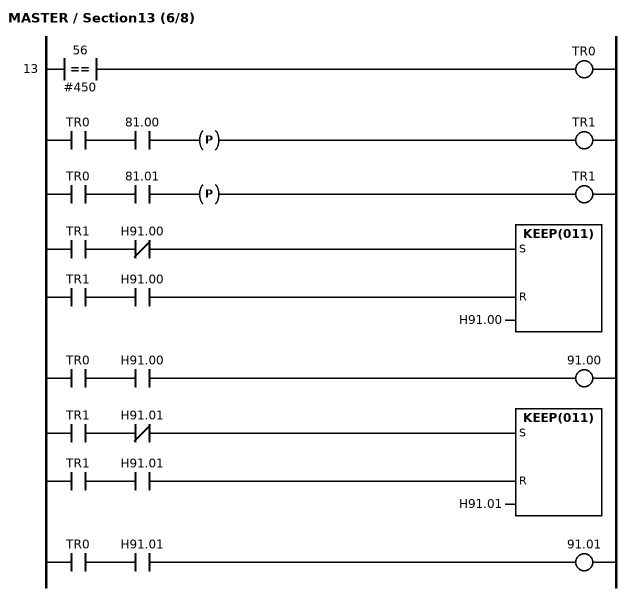
; [picture p48: MASTER / Section13, rungs 13-13]
; rung 13
LD=(300) 56 #450
OUT TR0
AND 81.00
UP(521)
OUT TR1
ANDNOT H91.00
LD TR1
AND H91.00
KEEP(011) H91.00
LD TR0
AND H91.00
OUT 91.00
LD TR0
AND 81.01
UP(521)
OUT TR1
ANDNOT H91.01
LD TR1
AND H91.01
KEEP(011) H91.01
LD TR0
AND H91.01
OUT 91.01

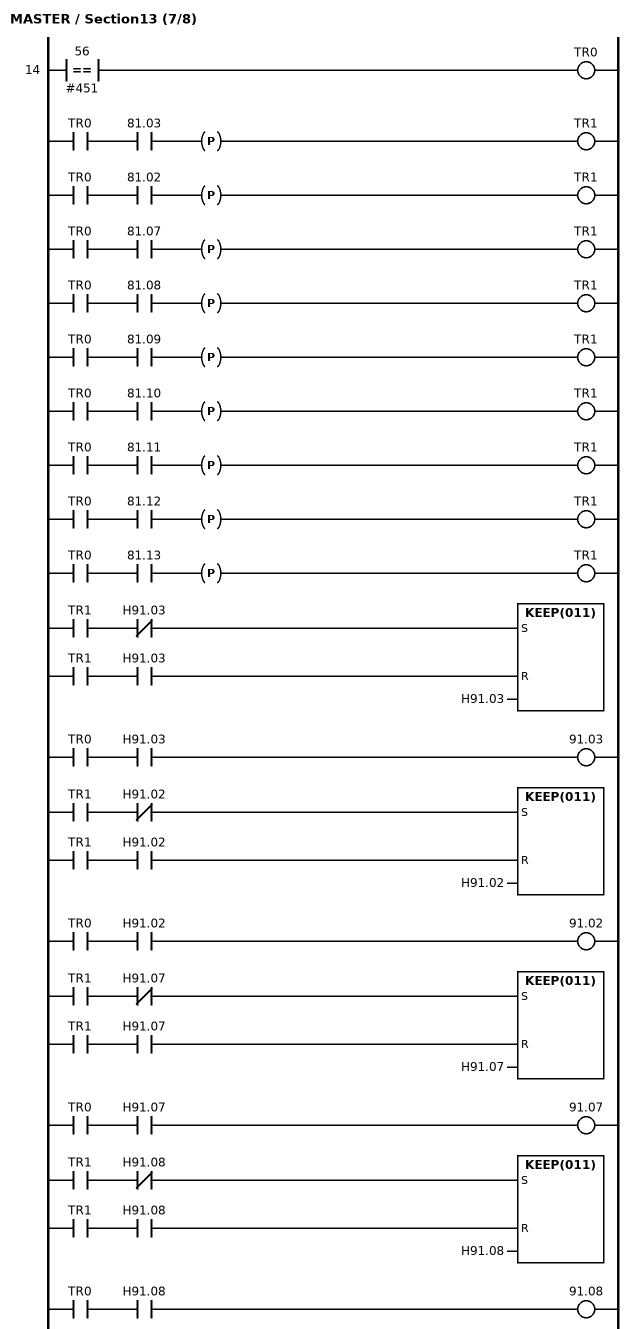

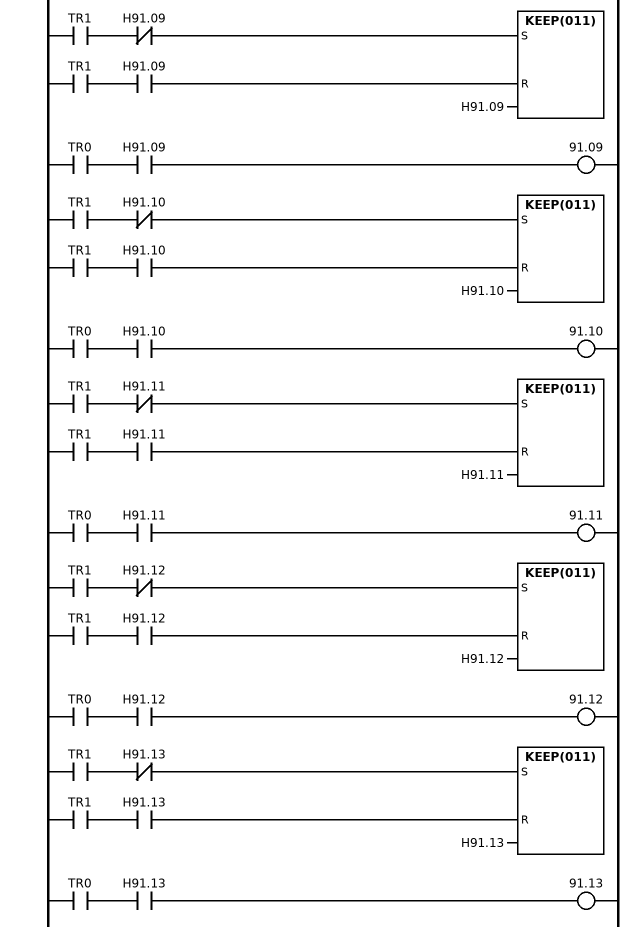
; rung 14
LD=(300) 56 #451
OUT TR0
AND 81.03
UP(521)
OUT TR1
ANDNOT H91.03
LD TR1
AND H91.03
KEEP(011) H91.03
LD TR0
AND H91.03
OUT 91.03
LD TR0
AND 81.02
UP(521)
OUT TR1
ANDNOT H91.02
LD TR1
AND H91.02
KEEP(011) H91.02
LD TR0
AND H91.02
OUT 91.02
LD TR0
AND 81.07
UP(521)
OUT TR1
ANDNOT H91.07
LD TR1
AND H91.07
KEEP(011) H91.07
LD TR0
AND H91.07
OUT 91.07
LD TR0
AND 81.08
UP(521)
OUT TR1
ANDNOT H91.08
LD TR1
AND H91.08
KEEP(011) H91.08
LD TR0
AND H91.08
OUT 91.08
LD TR0
AND 81.09
UP(521)
OUT TR1
ANDNOT H91.09
LD TR1
AND H91.09
KEEP(011) H91.09
LD TR0
AND H91.09
OUT 91.09
LD TR0
AND 81.10
UP(521)
OUT TR1
ANDNOT H91.10
LD TR1
AND H91.10
KEEP(011) H91.10
LD TR0
AND H91.10
OUT 91.10
LD TR0
AND 81.11
UP(521)
OUT TR1
ANDNOT H91.11
LD TR1
AND H91.11
KEEP(011) H91.11
LD TR0
AND H91.11
OUT 91.11
LD TR0
AND 81.12
UP(521)
OUT TR1
ANDNOT H91.12
LD TR1
AND H91.12
KEEP(011) H91.12
LD TR0
AND H91.12
OUT 91.12
LD TR0
AND 81.13
UP(521)
OUT TR1
ANDNOT H91.13
LD TR1
AND H91.13
KEEP(011) H91.13
LD TR0
AND H91.13
OUT 91.13

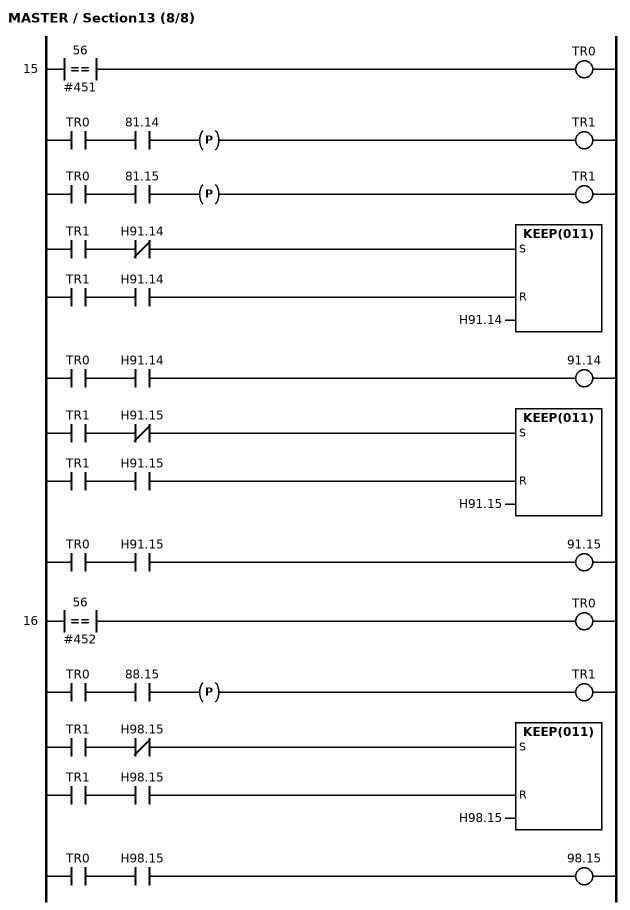
; rung 15
LD=(300) 56 #451
OUT TR0
AND 81.14
UP(521)
OUT TR1
ANDNOT H91.14
LD TR1
AND H91.14
KEEP(011) H91.14
LD TR0
AND H91.14
OUT 91.14
LD TR0
AND 81.15
UP(521)
OUT TR1
ANDNOT H91.15
LD TR1
AND H91.15
KEEP(011) H91.15
LD TR0
AND H91.15
OUT 91.15
; rung 16
LD=(300) 56 #452
OUT TR0
AND 88.15
UP(521)
OUT TR1
ANDNOT H98.15
LD TR1
AND H98.15
KEEP(011) H98.15
LD TR0
AND H98.15
OUT 98.15

### Section Section14

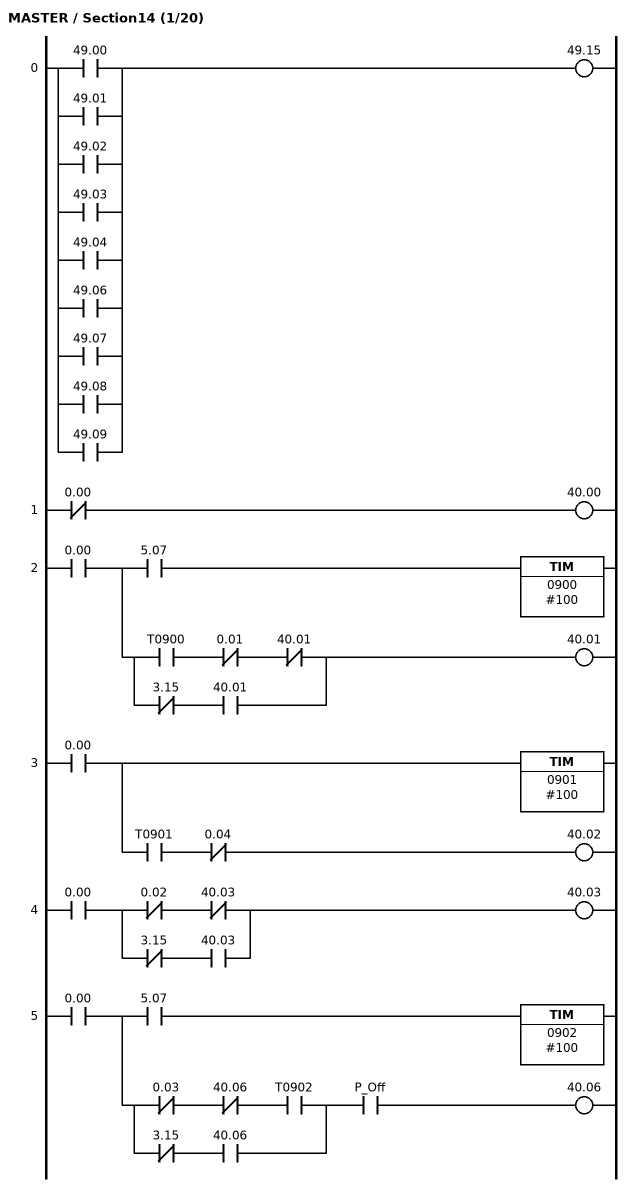
; rung 0
// R
LD 49.00
OR 49.01
OR 49.02
OR 49.03
OR 49.04
OR 49.06
OR 49.07
OR 49.08
OR 49.09
OUT 49.15
; rung 1
// R
LDNOT 0.00
OUT 40.00
; rung 2
// R
LD 0.00
OUT TR0
AND 5.07
TIM 0900 #100
LD TR0
LD T0900
ANDNOT 0.01
ANDNOT 40.01
LDNOT 3.15
AND 40.01
ORLD
ANDLD
OUT 40.01
; rung 3
// R
LD 0.00
TIM 0901 #100
AND T0901
ANDNOT 0.04
OUT 40.02
; rung 4
// R
LD 0.00
LDNOT 0.02
ANDNOT 40.03
LDNOT 3.15
AND 40.03
ORLD
ANDLD
OUT 40.03
; rung 5
// R
LD 0.00
OUT TR0
AND 5.07
TIM 0902 #100
LD TR0
LDNOT 0.03
ANDNOT 40.06
AND T0902
LDNOT 3.15
AND 40.06
ORLD
AND P_Off
ANDLD
OUT 40.06

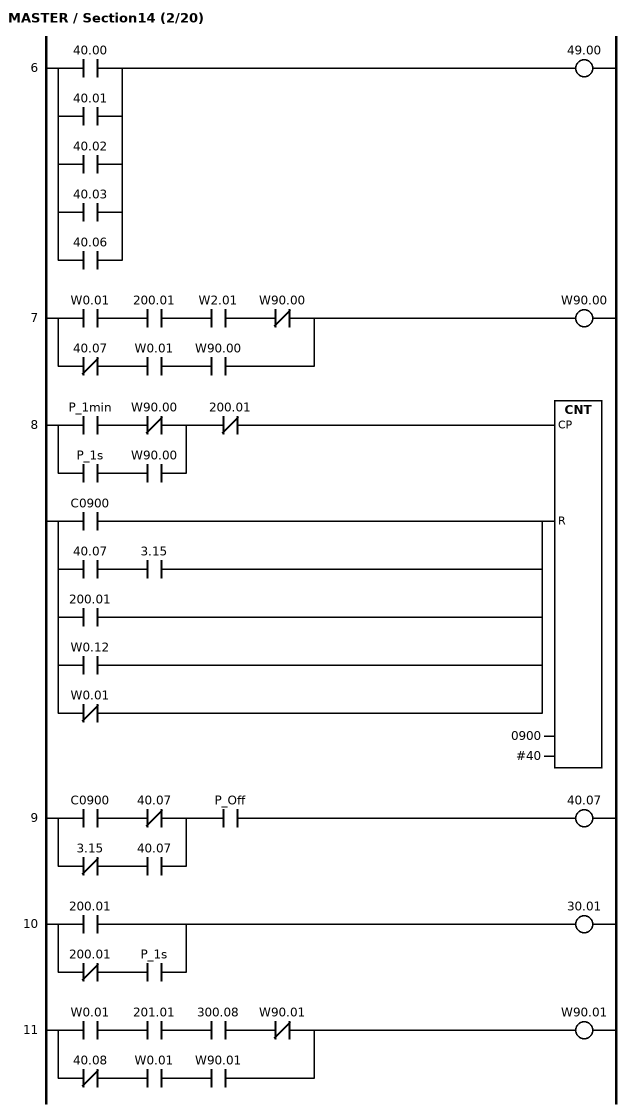
; rung 6
// R
LD 40.00
OR 40.01
OR 40.02
OR 40.03
OR 40.06
OUT 49.00
; rung 7
// R
LD W0.01
AND 200.01
AND W2.01
ANDNOT W90.00
LDNOT 40.07
AND W0.01
AND W90.00
ORLD
OUT W90.00
; rung 8
LD P_1min
ANDNOT W90.00
LD P_1s
AND W90.00
ORLD
ANDNOT 200.01
LD C0900
LD 40.07
AND 3.15
ORLD
OR 200.01
OR W0.12
ORNOT W0.01
CNT 0900 #40
; rung 9
LD C0900
ANDNOT 40.07
LDNOT 3.15
AND 40.07
ORLD
AND P_Off
OUT 40.07
; rung 10
LD 200.01
LDNOT 200.01
AND P_1s
ORLD
OUT 30.01
; rung 11
// R
LD W0.01
AND 201.01
AND 300.08
ANDNOT W90.01
LDNOT 40.08
AND W0.01
AND W90.01
ORLD
OUT W90.01

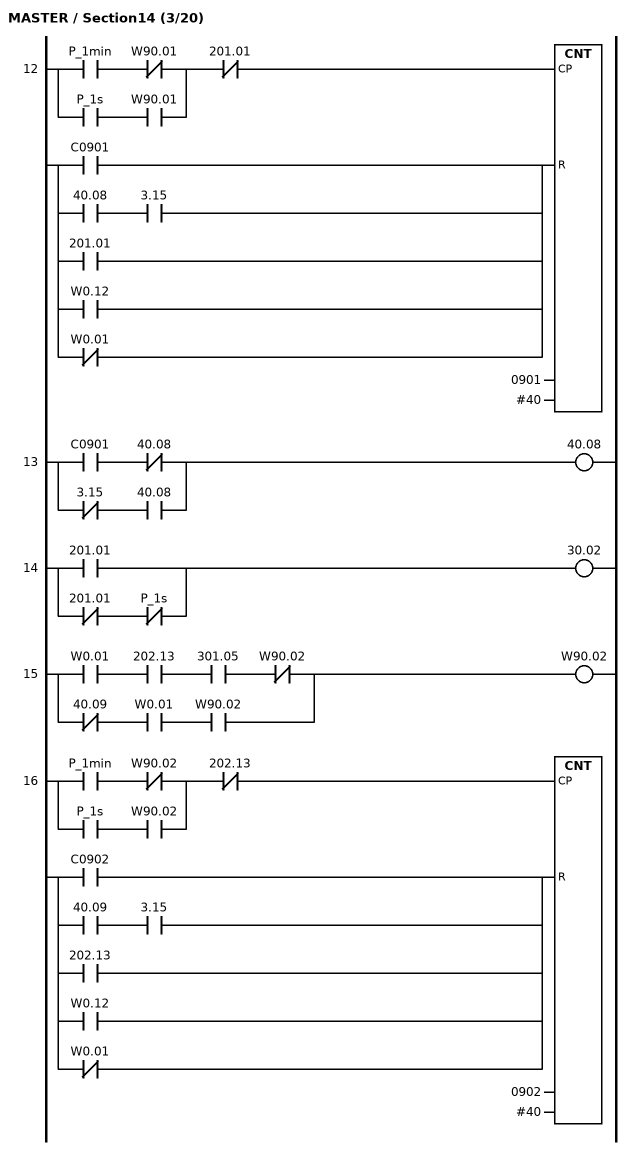
; rung 12
LD P_1min
ANDNOT W90.01
LD P_1s
AND W90.01
ORLD
ANDNOT 201.01
LD C0901
LD 40.08
AND 3.15
ORLD
OR 201.01
OR W0.12
ORNOT W0.01
CNT 0901 #40
; rung 13
LD C0901
ANDNOT 40.08
LDNOT 3.15
AND 40.08
ORLD
OUT 40.08
; rung 14
LD 201.01
LDNOT 201.01
ANDNOT P_1s
ORLD
OUT 30.02
; rung 15
// R
LD W0.01
AND 202.13
AND 301.05
ANDNOT W90.02
LDNOT 40.09
AND W0.01
AND W90.02
ORLD
OUT W90.02
; rung 16
LD P_1min
ANDNOT W90.02
LD P_1s
AND W90.02
ORLD
ANDNOT 202.13
LD C0902
LD 40.09
AND 3.15
ORLD
OR 202.13
OR W0.12
ORNOT W0.01
CNT 0902 #40

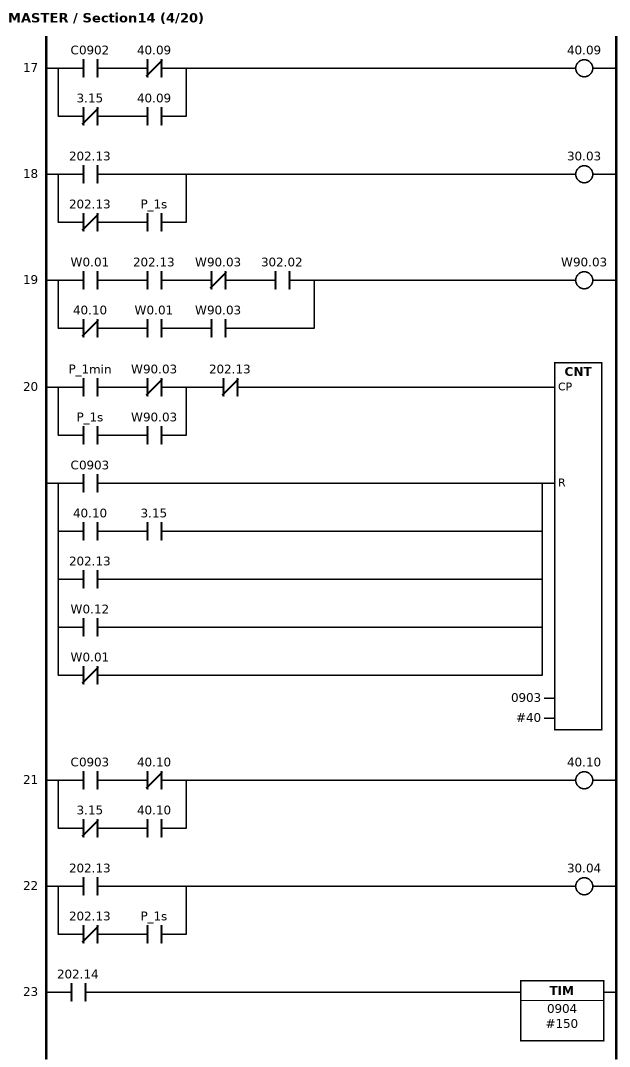
; rung 17
LD C0902
ANDNOT 40.09
LDNOT 3.15
AND 40.09
ORLD
OUT 40.09
; rung 18
LD 202.13
LDNOT 202.13
AND P_1s
ORLD
OUT 30.03
; rung 19
// R
LD W0.01
AND 202.13
ANDNOT W90.03
AND 302.02
LDNOT 40.10
AND W0.01
AND W90.03
ORLD
OUT W90.03
; rung 20
LD P_1min
ANDNOT W90.03
LD P_1s
AND W90.03
ORLD
ANDNOT 202.13
LD C0903
LD 40.10
AND 3.15
ORLD
OR 202.13
OR W0.12
ORNOT W0.01
CNT 0903 #40
; rung 21
LD C0903
ANDNOT 40.10
LDNOT 3.15
AND 40.10
ORLD
OUT 40.10
; rung 22
LD 202.13
LDNOT 202.13
AND P_1s
ORLD
OUT 30.04
; rung 23
LD 202.14
TIM 0904 #150

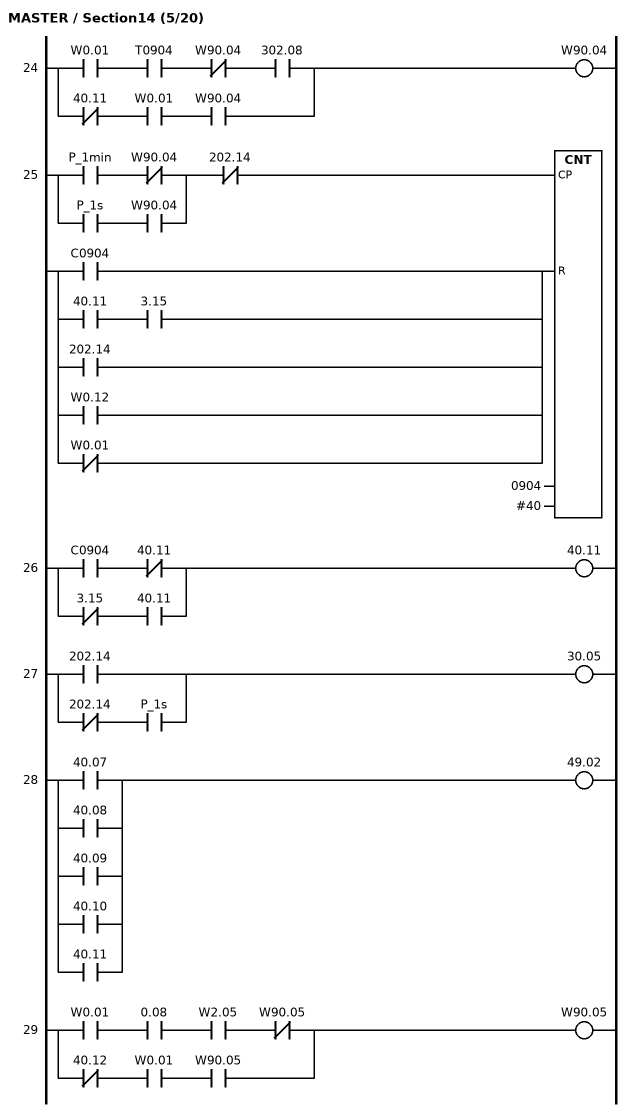
; rung 24
// R
LD W0.01
AND T0904
ANDNOT W90.04
AND 302.08
LDNOT 40.11
AND W0.01
AND W90.04
ORLD
OUT W90.04
; rung 25
LD P_1min
ANDNOT W90.04
LD P_1s
AND W90.04
ORLD
ANDNOT 202.14
LD C0904
LD 40.11
AND 3.15
ORLD
OR 202.14
OR W0.12
ORNOT W0.01
CNT 0904 #40
; rung 26
LD C0904
ANDNOT 40.11
LDNOT 3.15
AND 40.11
ORLD
OUT 40.11
; rung 27
LD 202.14
LDNOT 202.14
AND P_1s
ORLD
OUT 30.05
; rung 28
LD 40.07
OR 40.08
OR 40.09
OR 40.10
OR 40.11
OUT 49.02
; rung 29
// R
LD W0.01
AND 0.08
AND W2.05
ANDNOT W90.05
LDNOT 40.12
AND W0.01
AND W90.05
ORLD
OUT W90.05

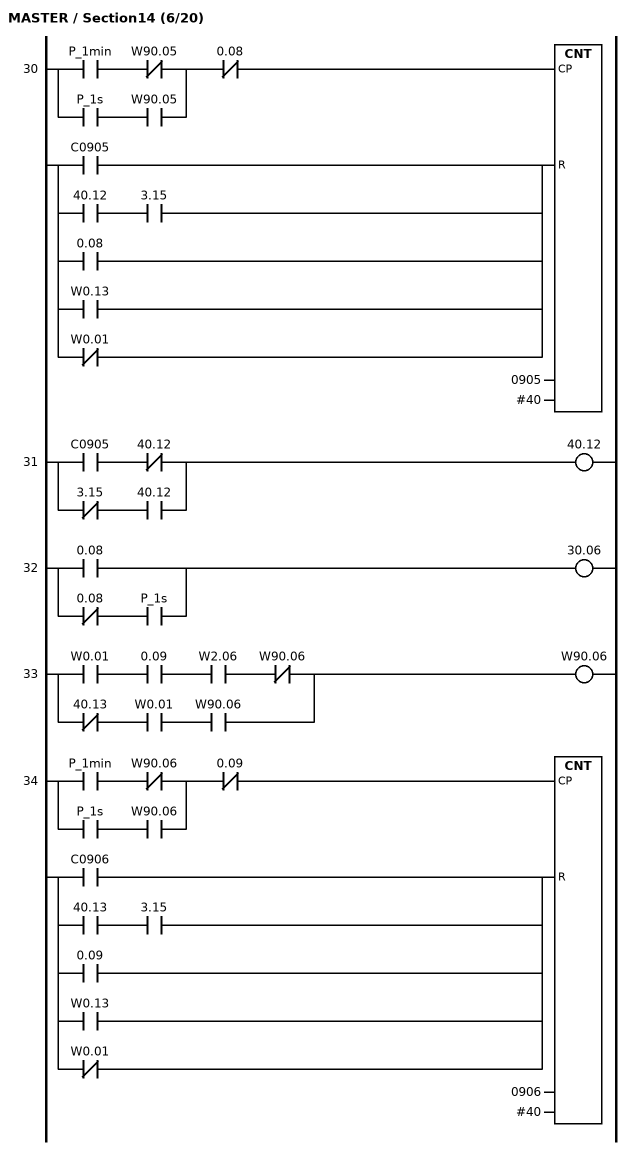
; rung 30
LD P_1min
ANDNOT W90.05
LD P_1s
AND W90.05
ORLD
ANDNOT 0.08
LD C0905
LD 40.12
AND 3.15
ORLD
OR 0.08
OR W0.13
ORNOT W0.01
CNT 0905 #40
; rung 31
LD C0905
ANDNOT 40.12
LDNOT 3.15
AND 40.12
ORLD
OUT 40.12
; rung 32
LD 0.08
LDNOT 0.08
AND P_1s
ORLD
OUT 30.06
; rung 33
// R
LD W0.01
AND 0.09
AND W2.06
ANDNOT W90.06
LDNOT 40.13
AND W0.01
AND W90.06
ORLD
OUT W90.06
; rung 34
LD P_1min
ANDNOT W90.06
LD P_1s
AND W90.06
ORLD
ANDNOT 0.09
LD C0906
LD 40.13
AND 3.15
ORLD
OR 0.09
OR W0.13
ORNOT W0.01
CNT 0906 #40

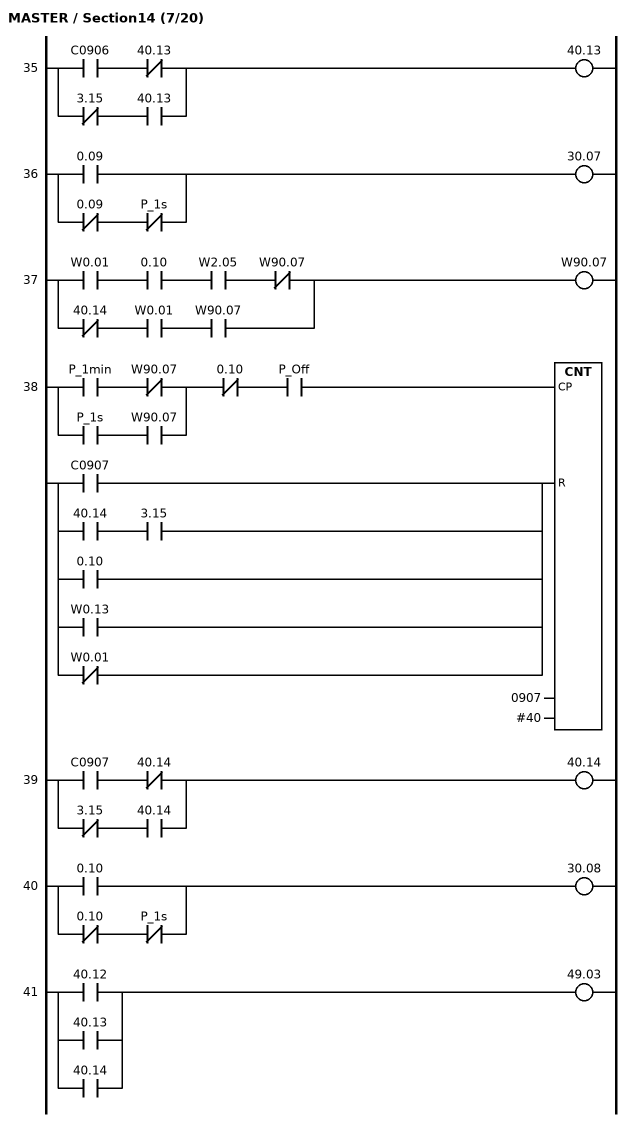
; rung 35
LD C0906
ANDNOT 40.13
LDNOT 3.15
AND 40.13
ORLD
OUT 40.13
; rung 36
LD 0.09
LDNOT 0.09
ANDNOT P_1s
ORLD
OUT 30.07
; rung 37
// R
LD W0.01
AND 0.10
AND W2.05
ANDNOT W90.07
LDNOT 40.14
AND W0.01
AND W90.07
ORLD
OUT W90.07
; rung 38
LD P_1min
ANDNOT W90.07
LD P_1s
AND W90.07
ORLD
ANDNOT 0.10
AND P_Off
LD C0907
LD 40.14
AND 3.15
ORLD
OR 0.10
OR W0.13
ORNOT W0.01
CNT 0907 #40
; rung 39
LD C0907
ANDNOT 40.14
LDNOT 3.15
AND 40.14
ORLD
OUT 40.14
; rung 40
LD 0.10
LDNOT 0.10
ANDNOT P_1s
ORLD
OUT 30.08
; rung 41
// R
LD 40.12
OR 40.13
OR 40.14
OUT 49.03

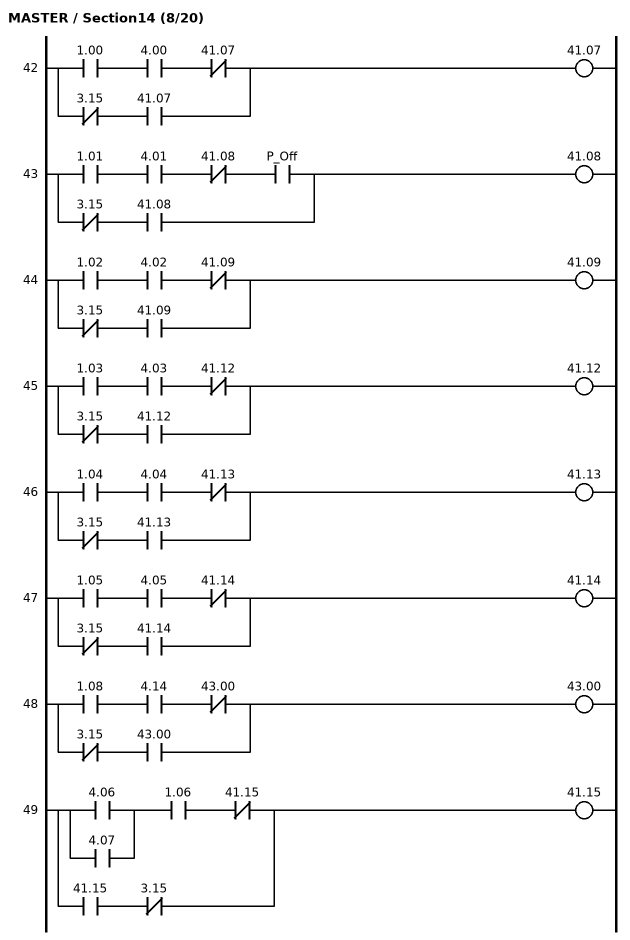
; rung 42
// R
LD 1.00
AND 4.00
ANDNOT 41.07
LDNOT 3.15
AND 41.07
ORLD
OUT 41.07
; rung 43
// R
LD 1.01
AND 4.01
ANDNOT 41.08
AND P_Off
LDNOT 3.15
AND 41.08
ORLD
OUT 41.08
; rung 44
// R
LD 1.02
AND 4.02
ANDNOT 41.09
LDNOT 3.15
AND 41.09
ORLD
OUT 41.09
; rung 45
// R
LD 1.03
AND 4.03
ANDNOT 41.12
LDNOT 3.15
AND 41.12
ORLD
OUT 41.12
; rung 46
// R
LD 1.04
AND 4.04
ANDNOT 41.13
LDNOT 3.15
AND 41.13
ORLD
OUT 41.13
; rung 47
// R
LD 1.05
AND 4.05
ANDNOT 41.14
LDNOT 3.15
AND 41.14
ORLD
OUT 41.14
; rung 48
// R
LD 1.08
AND 4.14
ANDNOT 43.00
LDNOT 3.15
AND 43.00
ORLD
OUT 43.00
; rung 49
// R
LD 4.06
OR 4.07
AND 1.06
ANDNOT 41.15
LD 41.15
ANDNOT 3.15
ORLD
OUT 41.15

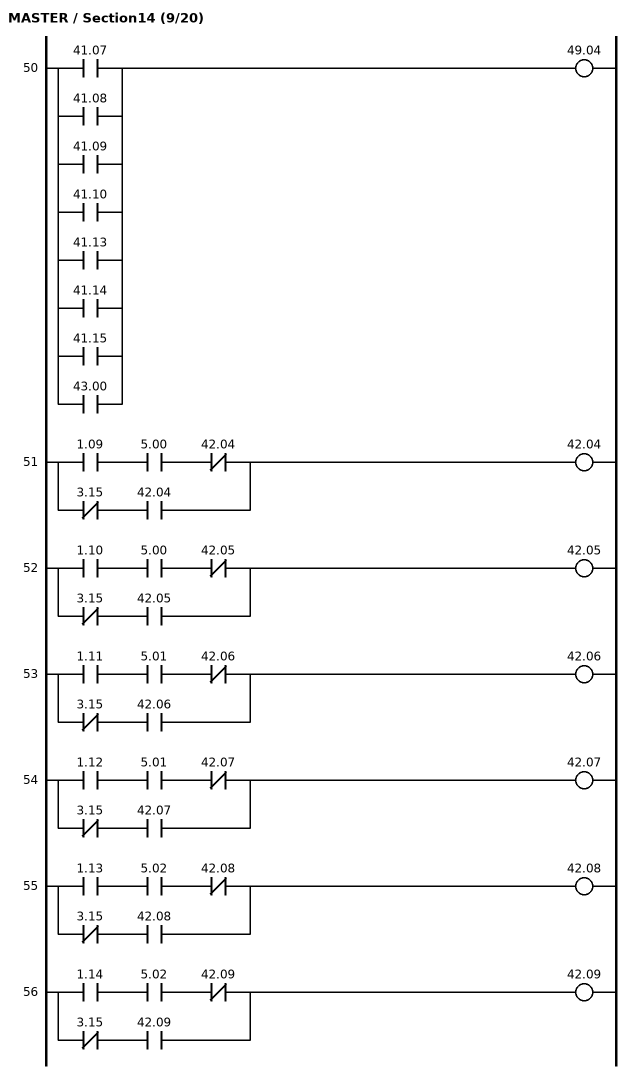
; rung 50
LD 41.07
OR 41.08
OR 41.09
OR 41.10
OR 41.13
OR 41.14
OR 41.15
OR 43.00
OUT 49.04
; rung 51
// R
LD 1.09
AND 5.00
ANDNOT 42.04
LDNOT 3.15
AND 42.04
ORLD
OUT 42.04
; rung 52
// R
LD 1.10
AND 5.00
ANDNOT 42.05
LDNOT 3.15
AND 42.05
ORLD
OUT 42.05
; rung 53
// R
LD 1.11
AND 5.01
ANDNOT 42.06
LDNOT 3.15
AND 42.06
ORLD
OUT 42.06
; rung 54
// R
LD 1.12
AND 5.01
ANDNOT 42.07
LDNOT 3.15
AND 42.07
ORLD
OUT 42.07
; rung 55
// R
LD 1.13
AND 5.02
ANDNOT 42.08
LDNOT 3.15
AND 42.08
ORLD
OUT 42.08
; rung 56
// R
LD 1.14
AND 5.02
ANDNOT 42.09
LDNOT 3.15
AND 42.09
ORLD
OUT 42.09

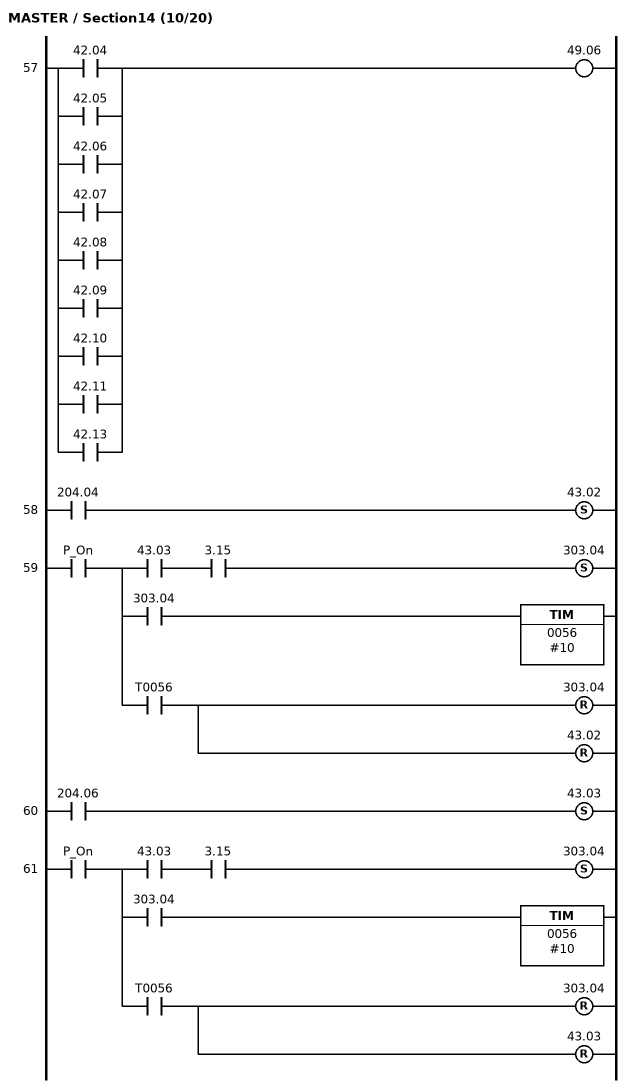
; rung 57
// R
LD 42.04
OR 42.05
OR 42.06
OR 42.07
OR 42.08
OR 42.09
OR 42.10
OR 42.11
OR 42.13
OUT 49.06
; rung 58
// R
LD 204.04
SET 43.02
; rung 59
LD P_On
OUT TR0
AND 43.03
AND 3.15
SET 303.04
LD TR0
AND 303.04
TIM 0056 #10
LD TR0
AND T0056
RSET 303.04
RSET 43.02
; rung 60
// R
LD 204.06
SET 43.03
; rung 61
LD P_On
OUT TR0
AND 43.03
AND 3.15
SET 303.04
LD TR0
AND 303.04
TIM 0056 #10
LD TR0
AND T0056
RSET 303.04
RSET 43.03

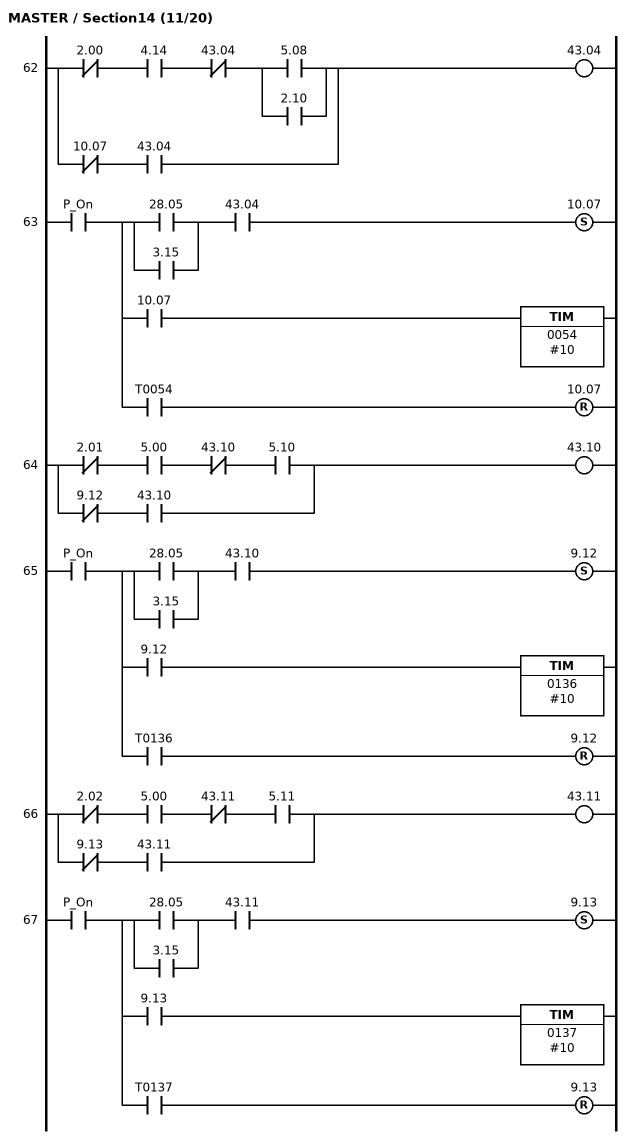
; rung 62
// R
LDNOT 2.00
AND 4.14
ANDNOT 43.04
LD 5.08
OR 2.10
ANDLD
LDNOT 10.07
AND 43.04
ORLD
OUT 43.04
; rung 63
LD P_On
OUT TR0
LD 28.05
OR 3.15
AND 43.04
ANDLD
SET 10.07
LD TR0
AND 10.07
TIM 0054 #10
LD TR0
AND T0054
RSET 10.07
; rung 64
// R
LDNOT 2.01
AND 5.00
ANDNOT 43.10
AND 5.10
LDNOT 9.12
AND 43.10
ORLD
OUT 43.10
; rung 65
LD P_On
OUT TR0
LD 28.05
OR 3.15
AND 43.10
ANDLD
SET 9.12
LD TR0
AND 9.12
TIM 0136 #10
LD TR0
AND T0136
RSET 9.12
; rung 66
// R
LDNOT 2.02
AND 5.00
ANDNOT 43.11
AND 5.11
LDNOT 9.13
AND 43.11
ORLD
OUT 43.11
; rung 67
LD P_On
OUT TR0
LD 28.05
OR 3.15
AND 43.11
ANDLD
SET 9.13
LD TR0
AND 9.13
TIM 0137 #10
LD TR0
AND T0137
RSET 9.13

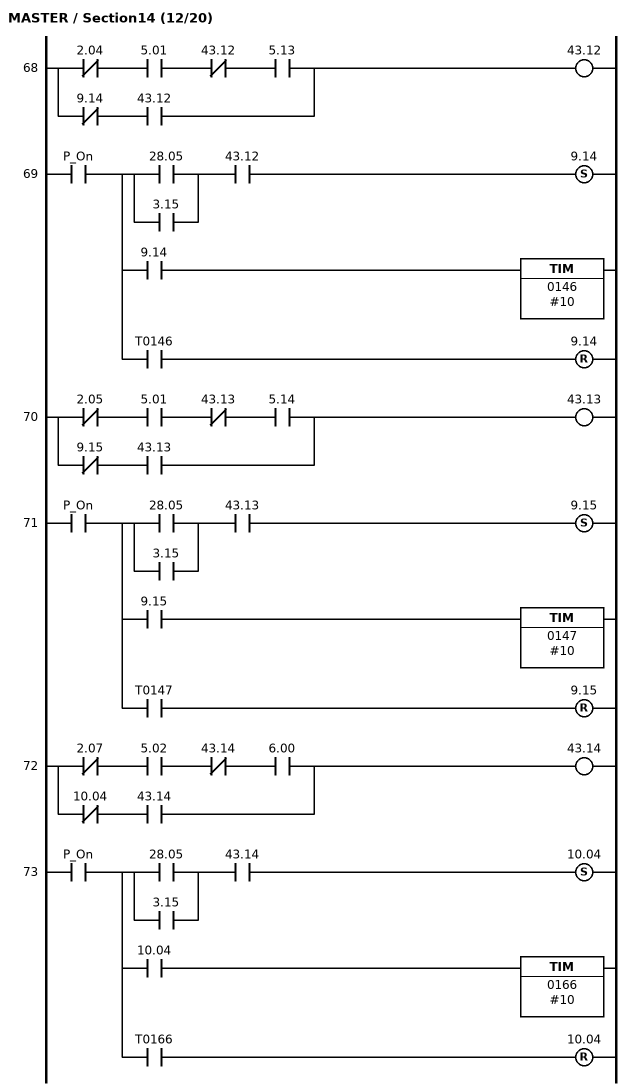
; rung 68
// R
LDNOT 2.04
AND 5.01
ANDNOT 43.12
AND 5.13
LDNOT 9.14
AND 43.12
ORLD
OUT 43.12
; rung 69
LD P_On
OUT TR0
LD 28.05
OR 3.15
AND 43.12
ANDLD
SET 9.14
LD TR0
AND 9.14
TIM 0146 #10
LD TR0
AND T0146
RSET 9.14
; rung 70
// R
LDNOT 2.05
AND 5.01
ANDNOT 43.13
AND 5.14
LDNOT 9.15
AND 43.13
ORLD
OUT 43.13
; rung 71
LD P_On
OUT TR0
LD 28.05
OR 3.15
AND 43.13
ANDLD
SET 9.15
LD TR0
AND 9.15
TIM 0147 #10
LD TR0
AND T0147
RSET 9.15
; rung 72
// R
LDNOT 2.07
AND 5.02
ANDNOT 43.14
AND 6.00
LDNOT 10.04
AND 43.14
ORLD
OUT 43.14
; rung 73
LD P_On
OUT TR0
LD 28.05
OR 3.15
AND 43.14
ANDLD
SET 10.04
LD TR0
AND 10.04
TIM 0166 #10
LD TR0
AND T0166
RSET 10.04

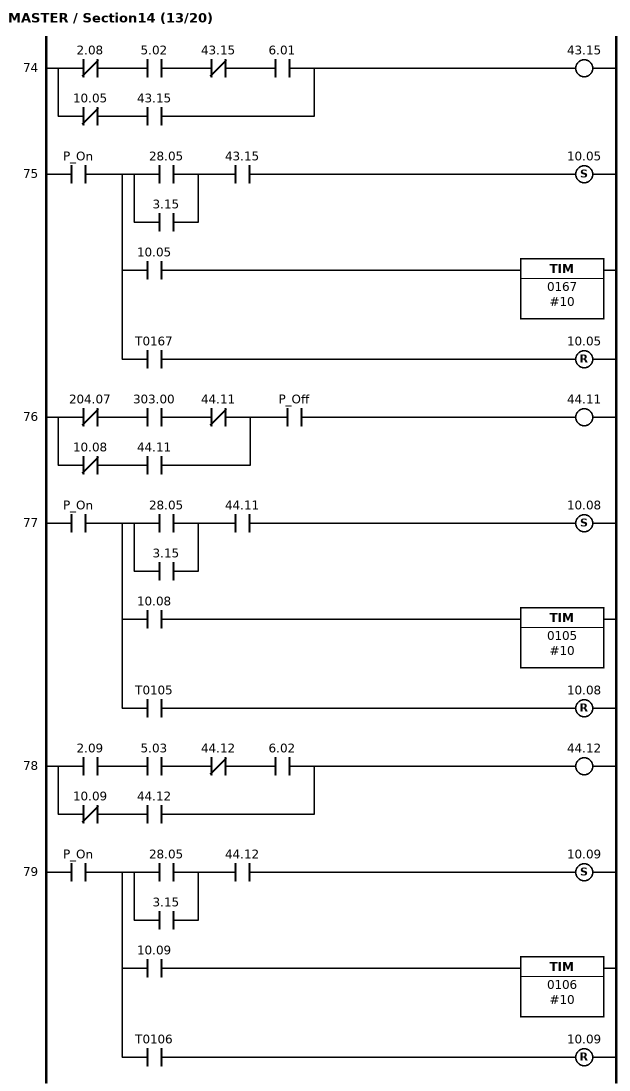
; rung 74
// R
LDNOT 2.08
AND 5.02
ANDNOT 43.15
AND 6.01
LDNOT 10.05
AND 43.15
ORLD
OUT 43.15
; rung 75
LD P_On
OUT TR0
LD 28.05
OR 3.15
AND 43.15
ANDLD
SET 10.05
LD TR0
AND 10.05
TIM 0167 #10
LD TR0
AND T0167
RSET 10.05
; rung 76
// R
LDNOT 204.07
AND 303.00
ANDNOT 44.11
LDNOT 10.08
AND 44.11
ORLD
AND P_Off
OUT 44.11
; rung 77
LD P_On
OUT TR0
LD 28.05
OR 3.15
AND 44.11
ANDLD
SET 10.08
LD TR0
AND 10.08
TIM 0105 #10
LD TR0
AND T0105
RSET 10.08
; rung 78
// R
LD 2.09
AND 5.03
ANDNOT 44.12
AND 6.02
LDNOT 10.09
AND 44.12
ORLD
OUT 44.12
; rung 79
LD P_On
OUT TR0
LD 28.05
OR 3.15
AND 44.12
ANDLD
SET 10.09
LD TR0
AND 10.09
TIM 0106 #10
LD TR0
AND T0106
RSET 10.09

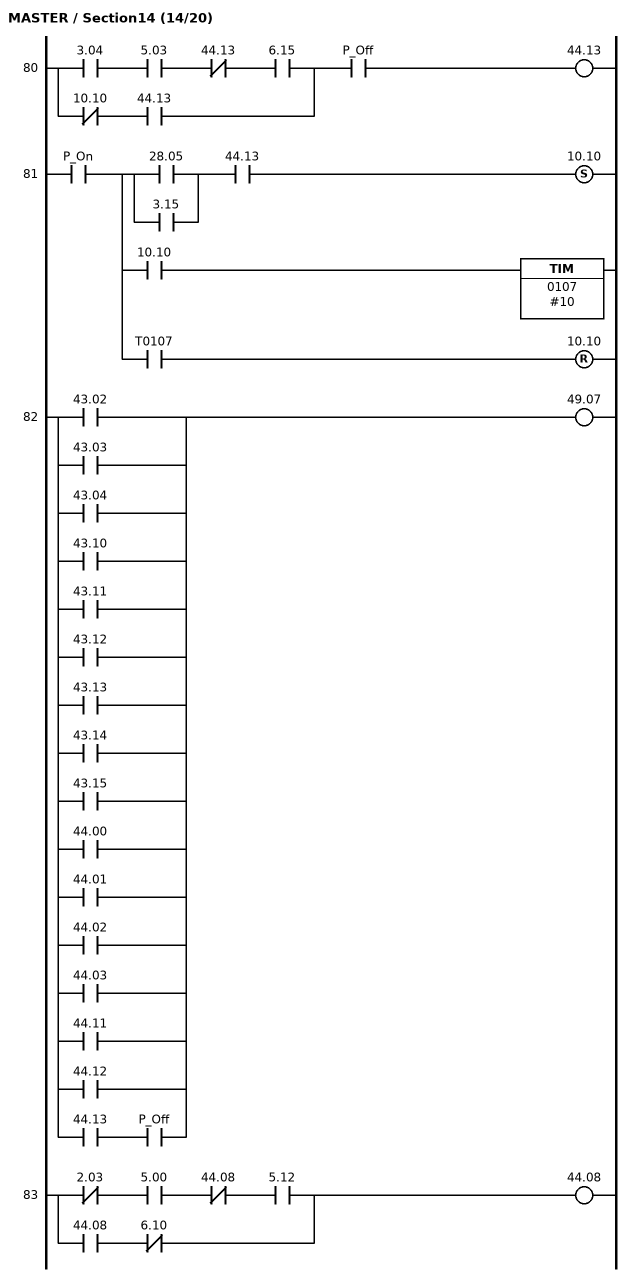
; rung 80
// R
LD 3.04
AND 5.03
ANDNOT 44.13
AND 6.15
LDNOT 10.10
AND 44.13
ORLD
AND P_Off
OUT 44.13
; rung 81
LD P_On
OUT TR0
LD 28.05
OR 3.15
AND 44.13
ANDLD
SET 10.10
LD TR0
AND 10.10
TIM 0107 #10
LD TR0
AND T0107
RSET 10.10
; rung 82
LD 43.02
OR 43.03
OR 43.04
OR 43.10
OR 43.11
OR 43.12
OR 43.13
OR 43.14
OR 43.15
OR 44.00
OR 44.01
OR 44.02
OR 44.03
OR 44.11
OR 44.12
LD 44.13
AND P_Off
ORLD
OUT 49.07
; rung 83
// R
LDNOT 2.03
AND 5.00
ANDNOT 44.08
AND 5.12
LD 44.08
ANDNOT 6.10
ORLD
OUT 44.08

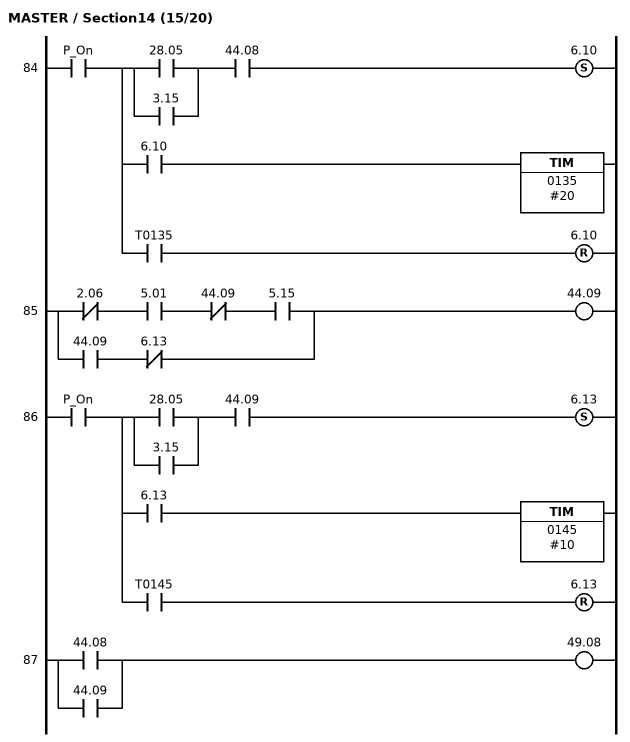
; rung 84
LD P_On
OUT TR0
LD 28.05
OR 3.15
AND 44.08
ANDLD
SET 6.10
LD TR0
AND 6.10
TIM 0135 #20
LD TR0
AND T0135
RSET 6.10
; rung 85
// R
LDNOT 2.06
AND 5.01
ANDNOT 44.09
AND 5.15
LD 44.09
ANDNOT 6.13
ORLD
OUT 44.09
; rung 86
LD P_On
OUT TR0
LD 28.05
OR 3.15
AND 44.09
ANDLD
SET 6.13
LD TR0
AND 6.13
TIM 0145 #10
LD TR0
AND T0145
RSET 6.13
; rung 87
// R
LD 44.08
OR 44.09
OUT 49.08

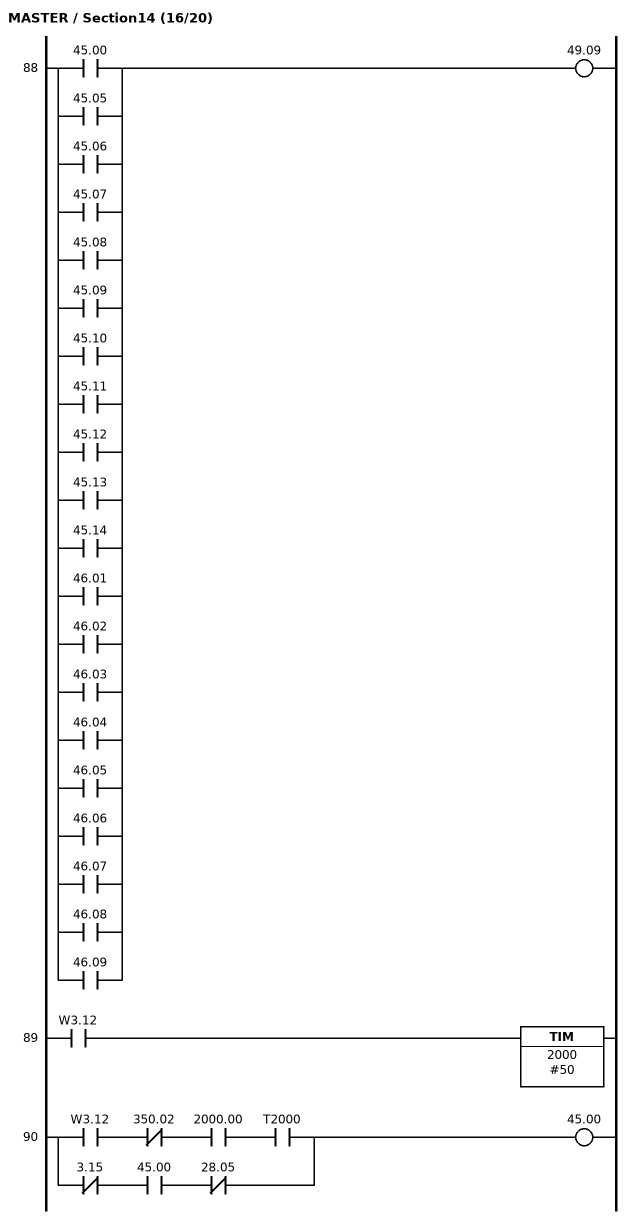
; rung 88
// R
LD 45.00
OR 45.05
OR 45.06
OR 45.07
OR 45.08
OR 45.09
OR 45.10
OR 45.11
OR 45.12
OR 45.13
OR 45.14
OR 46.01
OR 46.02
OR 46.03
OR 46.04
OR 46.05
OR 46.06
OR 46.07
OR 46.08
OR 46.09
OUT 49.09
; rung 89
// R
LD W3.12
TIM 2000 #50
; rung 90
// R
LD W3.12
ANDNOT 350.02
AND 2000.00
AND T2000
LDNOT 3.15
AND 45.00
ANDNOT 28.05
ORLD
OUT 45.00

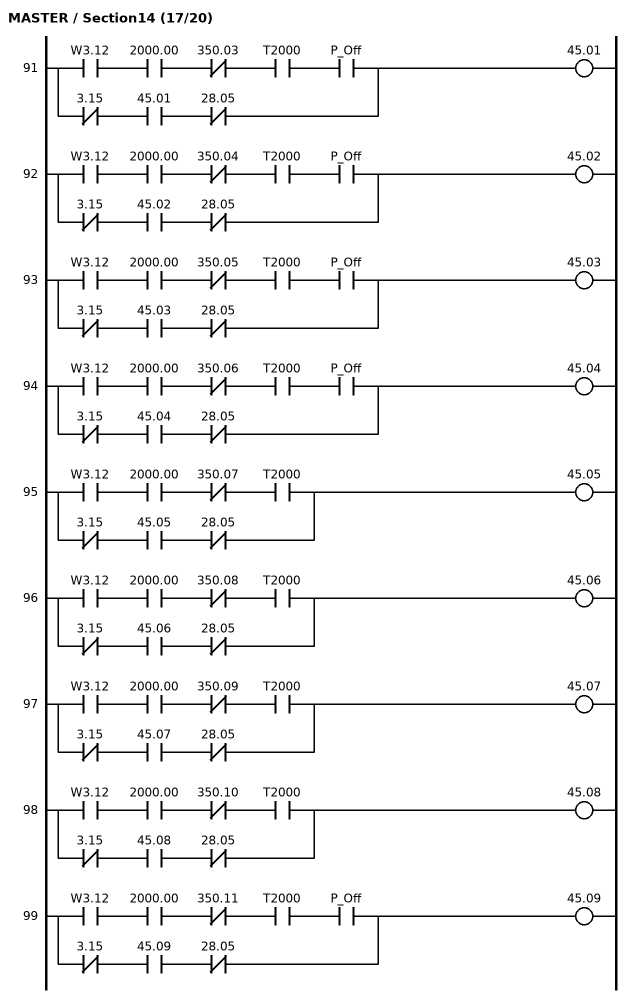
; rung 91
LD W3.12
AND 2000.00
ANDNOT 350.03
AND T2000
AND P_Off
LDNOT 3.15
AND 45.01
ANDNOT 28.05
ORLD
OUT 45.01
; rung 92
LD W3.12
AND 2000.00
ANDNOT 350.04
AND T2000
AND P_Off
LDNOT 3.15
AND 45.02
ANDNOT 28.05
ORLD
OUT 45.02
; rung 93
LD W3.12
AND 2000.00
ANDNOT 350.05
AND T2000
AND P_Off
LDNOT 3.15
AND 45.03
ANDNOT 28.05
ORLD
OUT 45.03
; rung 94
LD W3.12
AND 2000.00
ANDNOT 350.06
AND T2000
AND P_Off
LDNOT 3.15
AND 45.04
ANDNOT 28.05
ORLD
OUT 45.04
; rung 95
LD W3.12
AND 2000.00
ANDNOT 350.07
AND T2000
LDNOT 3.15
AND 45.05
ANDNOT 28.05
ORLD
OUT 45.05
; rung 96
LD W3.12
AND 2000.00
ANDNOT 350.08
AND T2000
LDNOT 3.15
AND 45.06
ANDNOT 28.05
ORLD
OUT 45.06
; rung 97
LD W3.12
AND 2000.00
ANDNOT 350.09
AND T2000
LDNOT 3.15
AND 45.07
ANDNOT 28.05
ORLD
OUT 45.07
; rung 98
LD W3.12
AND 2000.00
ANDNOT 350.10
AND T2000
LDNOT 3.15
AND 45.08
ANDNOT 28.05
ORLD
OUT 45.08
; rung 99
LD W3.12
AND 2000.00
ANDNOT 350.11
AND T2000
AND P_Off
LDNOT 3.15
AND 45.09
ANDNOT 28.05
ORLD
OUT 45.09

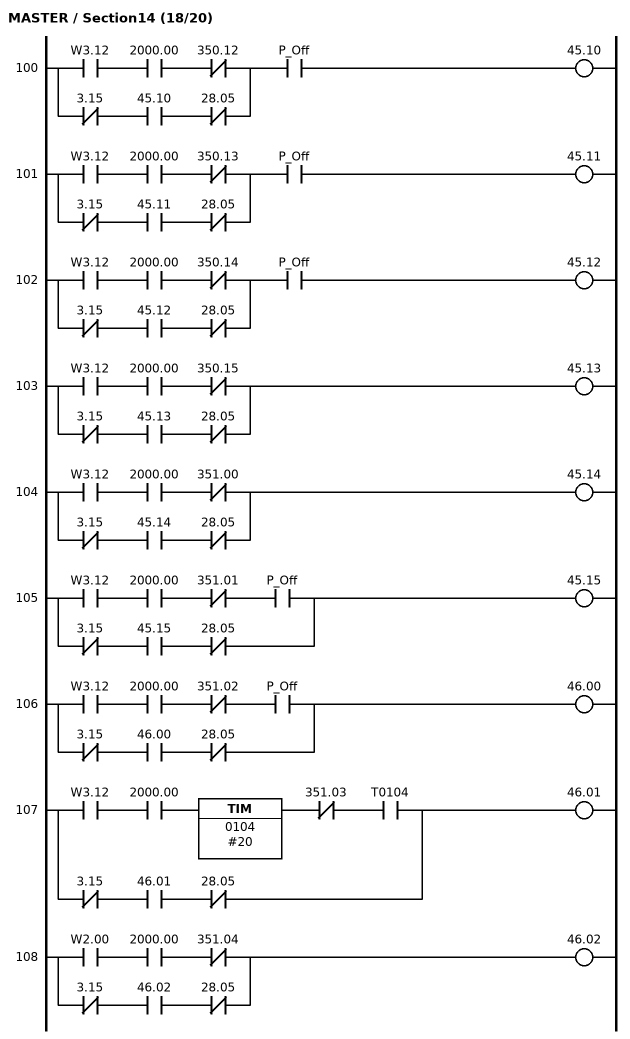
; rung 100
LD W3.12
AND 2000.00
ANDNOT 350.12
LDNOT 3.15
AND 45.10
ANDNOT 28.05
ORLD
AND P_Off
OUT 45.10
; rung 101
LD W3.12
AND 2000.00
ANDNOT 350.13
LDNOT 3.15
AND 45.11
ANDNOT 28.05
ORLD
AND P_Off
OUT 45.11
; rung 102
LD W3.12
AND 2000.00
ANDNOT 350.14
LDNOT 3.15
AND 45.12
ANDNOT 28.05
ORLD
AND P_Off
OUT 45.12
; rung 103
LD W3.12
AND 2000.00
ANDNOT 350.15
LDNOT 3.15
AND 45.13
ANDNOT 28.05
ORLD
OUT 45.13
; rung 104
LD W3.12
AND 2000.00
ANDNOT 351.00
LDNOT 3.15
AND 45.14
ANDNOT 28.05
ORLD
OUT 45.14
; rung 105
LD W3.12
AND 2000.00
ANDNOT 351.01
AND P_Off
LDNOT 3.15
AND 45.15
ANDNOT 28.05
ORLD
OUT 45.15
; rung 106
LD W3.12
AND 2000.00
ANDNOT 351.02
AND P_Off
LDNOT 3.15
AND 46.00
ANDNOT 28.05
ORLD
OUT 46.00
; rung 107
LD W3.12
AND 2000.00
TIM 0104 #20
ANDNOT 351.03
AND T0104
LDNOT 3.15
AND 46.01
ANDNOT 28.05
ORLD
OUT 46.01
; rung 108
LD W2.00
AND 2000.00
ANDNOT 351.04
LDNOT 3.15
AND 46.02
ANDNOT 28.05
ORLD
OUT 46.02

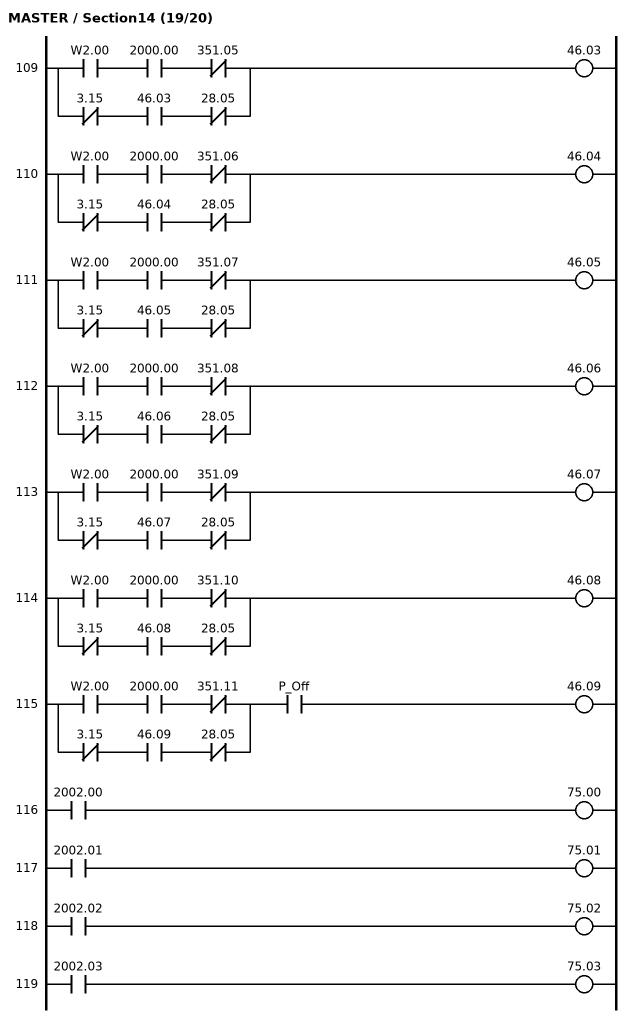
; rung 109
LD W2.00
AND 2000.00
ANDNOT 351.05
LDNOT 3.15
AND 46.03
ANDNOT 28.05
ORLD
OUT 46.03
; rung 110
LD W2.00
AND 2000.00
ANDNOT 351.06
LDNOT 3.15
AND 46.04
ANDNOT 28.05
ORLD
OUT 46.04
; rung 111
LD W2.00
AND 2000.00
ANDNOT 351.07
LDNOT 3.15
AND 46.05
ANDNOT 28.05
ORLD
OUT 46.05
; rung 112
LD W2.00
AND 2000.00
ANDNOT 351.08
LDNOT 3.15
AND 46.06
ANDNOT 28.05
ORLD
OUT 46.06
; rung 113
LD W2.00
AND 2000.00
ANDNOT 351.09
LDNOT 3.15
AND 46.07
ANDNOT 28.05
ORLD
OUT 46.07
; rung 114
LD W2.00
AND 2000.00
ANDNOT 351.10
LDNOT 3.15
AND 46.08
ANDNOT 28.05
ORLD
OUT 46.08
; rung 115
LD W2.00
AND 2000.00
ANDNOT 351.11
LDNOT 3.15
AND 46.09
ANDNOT 28.05
ORLD
AND P_Off
OUT 46.09
; rung 116
LD 2002.00
OUT 75.00
; rung 117
LD 2002.01
OUT 75.01
; rung 118
LD 2002.02
OUT 75.02
; rung 119
LD 2002.03
OUT 75.03

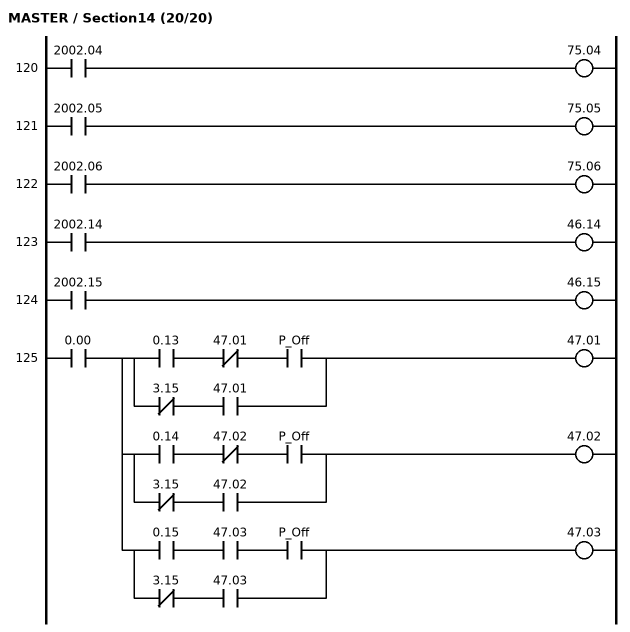
; rung 120
LD 2002.04
OUT 75.04
; rung 121
LD 2002.05
OUT 75.05
; rung 122
LD 2002.06
OUT 75.06
; rung 123
LD 2002.14
OUT 46.14
; rung 124
LD 2002.15
OUT 46.15
; rung 125
LD 0.00
OUT TR0
LD 0.13
ANDNOT 47.01
AND P_Off
LDNOT 3.15
AND 47.01
ORLD
ANDLD
OUT 47.01
LD TR0
LD 0.14
ANDNOT 47.02
AND P_Off
LDNOT 3.15
AND 47.02
ORLD
ANDLD
OUT 47.02
LD TR0
LD 0.15
AND 47.03
AND P_Off
LDNOT 3.15
AND 47.03
ORLD
ANDLD
OUT 47.03

### Section Section15

